Staubli VAL3: PlasticMain.dtx

num nPLCRestartCnt
string programList
string sTaskName[3]
  [0] = "PLC_Main"
  [1] = "MP_MainPRG"
  [2] = "SR_HomeReturn"
string sVersion
string sBuildNumber
bool bFirstLoad = true
bool bStartUp
bool homeFlag
bool overrun
string sRawList
string sCopyRight = "Plastics (C) 2006-2011 V"
